FUNCTION_BLOCK FB_ISKRA_T5
// FB Utilisée uniquement pour motherfucking ISKRA de mes couilles.... 
// 
VAR_INPUT

	WORD_WEAK		: WORD;				// Strong Word. Word to consider if size equals 1.
	WORD_STRONG		: WORD;
END_VAR
VAR_OUTPUT
	VAR_OUT			: REAL;
END_VAR
VAR
	FullWord		: DWORD;
	ValExp			: SINT;
	ValCorps		: UDINT;
END_VAR


FullWord := SHL(WORD_TO_DWORD(WORD_STRONG), 16) OR WORD_Weak;

ValExp := BYTE_TO_SINT(DWORD_TO_BYTE(SHR(FullWord, 24)));
ValCorps := DWORD_TO_UDINT(SHR(SHL(FullWord, 8),8));

VAR_OUT :=  ValCorps*EXPT(10, ValExp);

END_FUNCTION_BLOCK

(* stored: Version 1.1.0.1, ProductVersion 3.1.4024.6
   POU FB_ISKRA_T5: Id {62e1f687-6767-44b2-826d-4608af9ebb0b}, SpecialFunc None *)
